// TIA Portal project "COLOUR DETECTION" (V15)
// Vorlageprojekt für das Buch mit Zielsystem S7-1200

(* hardware
DEVICE "S7-1200-Station_1"  S7-1200 Station
   slot 0: "Baugruppenträger_0"  Rack  V1.0
   slot 1: "PLC_1"  CPU 1211C DC/DC/DC  6ES7 211-1AE40-0XB0  V4.1
*)

// ===== PLC "PLC_1"  CPU 1211C DC/DC/DC =====

VAR_GLOBAL   // PLC tag table "Standard-Variablentabelle"
   "MAIN BELT" AT %A0.0 : Bool;
   "START" AT %E0.0 : Bool;
   "STOP" AT %E0.1 : Bool;
   "BELT 2" AT %Q0.2 : Bool;
   "SENSOR 1" AT %I0.2 : Bool;
   "BELT 3" AT %Q0.3 : Bool;
   "CURVED BELT" AT %Q0.4 : Bool;
   "PUSHER 1" AT %Q0.5 : Bool;
   "BACK PUSHER 1" AT %I0.4 : Bool;
   "BELT 1" AT %Q0.1 : Bool;
   "FRONT PUSHER 1" AT %I0.6 : Bool;
   "SENSOR 2" AT %I0.3 : Bool;
   "M 0" AT %M0.0 : Bool;
   "PUSHER 2" AT %Q0.6 : Bool;
   "BACK PUSHER 2" AT %I0.5 : Bool;
   "FRONT PUSHER 2" AT %I0.7 : Bool;
END_VAR

FUNCTION "MHJ-PLC-Lab-Function-S71200" : Void   // FC9000, SCL
{ S7_Optimized_Access := 'TRUE' }
VERSION : 0.1
   VAR_TEMP
      rdTimeReturn : Int;
      outputTime : DTL;
      SyncVal : Byte;
      forVal : Int;
      forVal_2 : Int;
      Value : Byte;
   END_VAR
   VAR CONSTANT
      CompVal : Byte := 16#34;
      Value_01 : Byte := 16#11;
      Value_01_DW : DWord := 16#A165_D992;
      Value_02_DW : DWord := 16#58BE_4401;
   END_VAR
BEGIN

   #Value:=PEEK(area := 16#82,
        dbNumber := 0,
        byteOffset := 511);
   #Value := #Value + 1;

   POKE(area := 16#82,
        dbNumber := 0,
        byteOffset := 511,
        value := #Value);

   POKE(area:=16#81,
        dbNumber:=0,
        byteOffset:=1016,
        value:=#Value_01_DW);
   POKE(area := 16#81,
        dbNumber := 0,
        byteOffset := 1020,
        value := #Value_02_DW);

   POKE(area := 16#81,
        dbNumber := 0,
        byteOffset := 511,
        value := B#16#00);

   FOR #forVal := 0 TO 120 DO
       FOR #forVal_2:=0 TO 10 DO
           #rdTimeReturn:=RD_SYS_T(#outputTime);
           #rdTimeReturn := WR_SYS_T(#outputTime);
           #rdTimeReturn := RD_SYS_T(#outputTime);
           #rdTimeReturn := WR_SYS_T(#outputTime);
       END_FOR;
       #SyncVal:= PEEK(area := 16#81,
                      dbNumber := 0,
                      byteOffset := 511);
       IF #SyncVal = #CompVal THEN
          GOTO M_1;
       END_IF;
   END_FOR;
   RETURN;

   M_1:
   POKE(area := 16#81,
        dbNumber := 0,
        byteOffset := 511,
        value := B#16#0);
END_FUNCTION

ORGANIZATION_BLOCK "Main"   // OB1, LAD, ProgramCycle
TITLE = "Main Program Sweep (Cycle)"
{ S7_Optimized_Access := 'TRUE' }
VERSION : 0.1
   VAR_INPUT
      Initial_Call : Bool;   // Initial call of this OB
      Remanence : Bool;   // =True, if remanent data are available
   END_VAR
BEGIN

REGION Network 1: Konnektierungsbaustein für PLC-Lab
   // Im Netzwerk 1 wird der Konnektierungsbaustein für PLC-Lab aufgerufen.
   // Dieser Aufruf darf nicht entfernt werden!
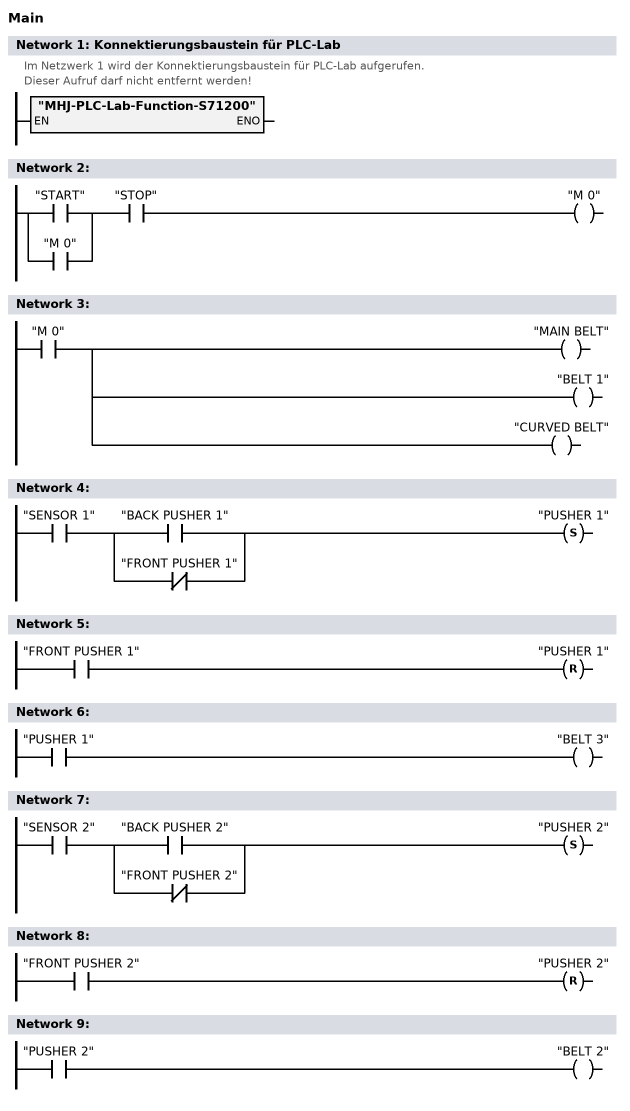
   RUNG wire#powerrail
      "MHJ-PLC-Lab-Function-S71200"()
   END_RUNG
   // the same network as SCL:
   "MHJ-PLC-Lab-Function-S71200"();
END_REGION

REGION Network 2
   RUNG wire#powerrail
      Contact( "START" )
      wire#w1
      Contact( "STOP" )
      Coil( "M 0" )
   END_RUNG
   RUNG wire#powerrail
      Contact( "M 0" )
   END_RUNG wire#w1
   // the same network as SCL:
   "M 0" := ("START" OR "M 0") AND "STOP";
END_REGION

REGION Network 3
   RUNG wire#powerrail
      Contact( "M 0" )
      wire#w1
      Coil( "MAIN BELT" )
   END_RUNG
   RUNG wire#w1
      Coil( "BELT 1" )
   END_RUNG
   RUNG wire#w1
      Coil( "CURVED BELT" )
   END_RUNG
   // the same network as SCL:
   "MAIN BELT" := "M 0";
   "BELT 1" := "M 0";
   "CURVED BELT" := "M 0";
END_REGION

REGION Network 4
   RUNG wire#powerrail
      Contact( "SENSOR 1" )
      wire#w1
      Contact( "BACK PUSHER 1" )
      wire#w2
      S_Coil( "PUSHER 1" )
   END_RUNG
   RUNG wire#w1
      I_Contact( "FRONT PUSHER 1" )
   END_RUNG wire#w2
   // the same network as SCL:
   IF "SENSOR 1" AND ("BACK PUSHER 1" OR NOT "FRONT PUSHER 1") THEN "PUSHER 1" := TRUE; END_IF;
END_REGION

REGION Network 5
   RUNG wire#powerrail
      Contact( "FRONT PUSHER 1" )
      R_Coil( "PUSHER 1" )
   END_RUNG
   // the same network as SCL:
   IF "FRONT PUSHER 1" THEN "PUSHER 1" := FALSE; END_IF;
END_REGION

REGION Network 6
   RUNG wire#powerrail
      Contact( "PUSHER 1" )
      Coil( "BELT 3" )
   END_RUNG
   // the same network as SCL:
   "BELT 3" := "PUSHER 1";
END_REGION

REGION Network 7
   RUNG wire#powerrail
      Contact( "SENSOR 2" )
      wire#w1
      Contact( "BACK PUSHER 2" )
      wire#w2
      S_Coil( "PUSHER 2" )
   END_RUNG
   RUNG wire#w1
      I_Contact( "FRONT PUSHER 2" )
   END_RUNG wire#w2
   // the same network as SCL:
   IF "SENSOR 2" AND ("BACK PUSHER 2" OR NOT "FRONT PUSHER 2") THEN "PUSHER 2" := TRUE; END_IF;
END_REGION

REGION Network 8
   RUNG wire#powerrail
      Contact( "FRONT PUSHER 2" )
      R_Coil( "PUSHER 2" )
   END_RUNG
   // the same network as SCL:
   IF "FRONT PUSHER 2" THEN "PUSHER 2" := FALSE; END_IF;
END_REGION

REGION Network 9
   RUNG wire#powerrail
      Contact( "PUSHER 2" )
      Coil( "BELT 2" )
   END_RUNG
   // the same network as SCL:
   "BELT 2" := "PUSHER 2";
END_REGION
END_ORGANIZATION_BLOCK